SUBAPPLICATION ASR2_DELAY_SUB (* ASR2_DELAY mit fest verdrahteten Verzoegerungszeiten (Franz: 'da jetzt Zeiten einbauen, einfach Fix mal. 2s oder so. Rein wie rauswaerts') - alle 4 Zeiten (SET/RESET x Vorwaerts/Rueckwaerts) fest auf T#2s, ueber initval_ATM initialisiert. STOP_* pass-through, optional von aussen verdrahtbar. *)
  (* Standard: 61499-2 *)
  (* Version 1.1, 2026-09-17, Franz Höpfinger, Meisterschulen am Ostbahnhof, Zeiten ergaenzt (Franz: '2s oder so, rein wie rauswaerts'): 4x initval_ATM (T#2s) auf PT_SET_FWD/PT_SET_BWD/PT_RESET_FWD/PT_RESET_BWD verdrahtet - Platzhalter-Fixwert, kein funktionale Vorgabe, spaeter parametrierbar falls noetig. STOP_SET_FWD/STOP_SET_BWD/STOP_RESET_FWD/STOP_RESET_BWD als Pass-through-Sockets ergaenzt (analog CHAIN_OUT), unverdrahtet lassen wenn nicht gebraucht. *)
  (* Version 1.0, 2026-09-17, franz *)
  PACKAGE MyLib::sys;
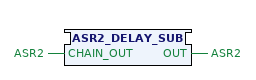
  SOCKETS
    CHAIN_OUT : adapter::types::bidirectional::ASR2;
  END_SOCKETS
  PLUGS
    OUT : adapter::types::bidirectional::ASR2;
  END_PLUGS
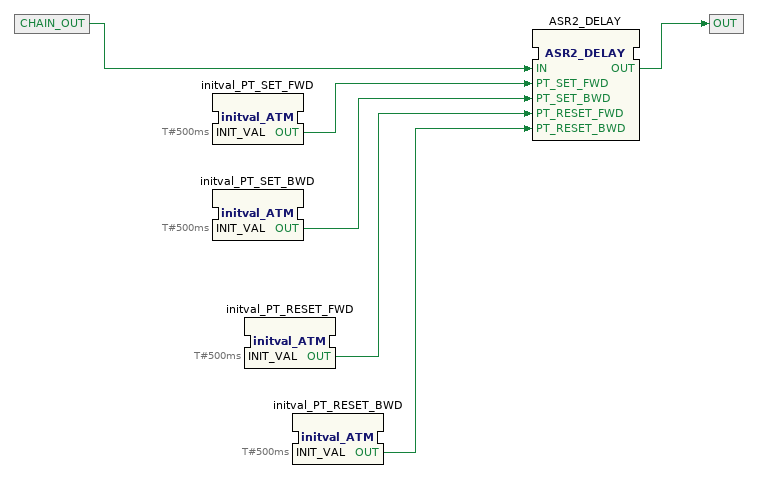
  FBS
    ASR2_DELAY : adapter::events::bidirectional::ASR2_DELAY;
    initval_PT_SET_FWD : adapter::types::unidirectional::ATM::initval::initval_ATM(INIT_VAL := T#500ms);
    initval_PT_SET_BWD : adapter::types::unidirectional::ATM::initval::initval_ATM(INIT_VAL := T#500ms);
    initval_PT_RESET_FWD : adapter::types::unidirectional::ATM::initval::initval_ATM(INIT_VAL := T#500ms);
    initval_PT_RESET_BWD : adapter::types::unidirectional::ATM::initval::initval_ATM(INIT_VAL := T#500ms);
  END_FBS
  ADAPTER_CONNECTIONS
    CHAIN_OUT TO ASR2_DELAY.IN;
    ASR2_DELAY.OUT TO OUT;
    initval_PT_SET_FWD.OUT TO ASR2_DELAY.PT_SET_FWD;
    initval_PT_SET_BWD.OUT TO ASR2_DELAY.PT_SET_BWD;
    initval_PT_RESET_FWD.OUT TO ASR2_DELAY.PT_RESET_FWD;
    initval_PT_RESET_BWD.OUT TO ASR2_DELAY.PT_RESET_BWD;
  END_CONNECTIONS
END_SUBAPPLICATION
